// TIA Portal V16 export
// export: Created 2022-11-14T17:35:43.5789192Z, ExportSetting WithDefaults, DisplayName Totally Integrated Automation Portal, DisplayVersion V16, DisplayName TIA Portal Version Control Interface, DisplayVersion V16, DisplayName TIA Portal Openness, DisplayVersion V16, DisplayName STEP 7 Professional, DisplayVersion V16, DisplayName STEP 7 Safety, DisplayVersion V16, DisplayName WinCC Advanced, DisplayVersion V16
DATA_BLOCK "Modbus_DB"   // DB28
VERSION : 0.1
// stored: AutoNumber false, InstanceOfName Modbus, InstanceOfType FB
"Modbus"
   // VAR_INPUT
   //    BAUDRATE : UDInt;
   //    HW_ID : PORT;
   //    RESP_TO : UInt;
   //    CYCLIC_PROCESSING : Bool;
   //    MB_ADDR : UInt;
   //    DATA_AD_R : UDInt;
   //    DATA_AD_W : UDInt;
   //    DATA_LEN_R : UInt;
   //    DATA_LEN_W : UInt;
   //    ReadOnly : Bool;
   // END_VAR
   // VAR_OUTPUT
   //    ERROR : Bool;
   //    ERROR_INFO : Struct
   //       drive_number : USInt;
   //       "step" : USInt;
   //       STATUS : Word;
   //    END_STRUCT;
   // END_VAR
   // VAR_IN_OUT
   //    ReadDone_0 : Bool;
   //    DT_PTR_IN : Variant;
   //    DT_PTR_OUT : Variant;
   // END_VAR
   // VAR
   //    drive_index : USInt;
   //    "step" : USInt;
   //    REQ : Bool;
   //    extended_restart : Bool;
   //    start_internal : Bool;
   //    MB_COMM_LOAD_Instance { S7_SetPoint := 'True'} : MB_COMM_LOAD;
   //    MB_MASTER_Instance { S7_SetPoint := 'True'} : MB_MASTER;
   // END_VAR
BEGIN
END_DATA_BLOCK
